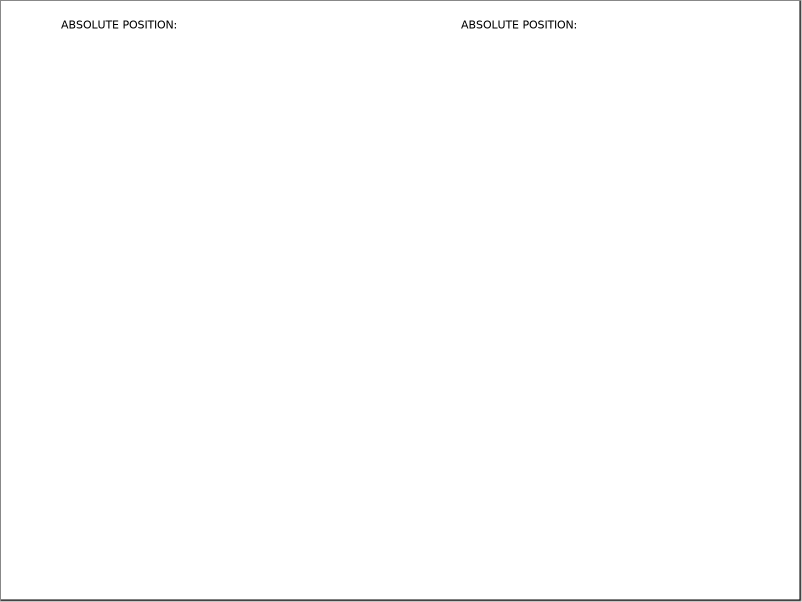
VISUALIZATION F51_Cam_Exchange  // 802x602
    Rectangle (0,0 800x600)
    Label (10,10 170x30), "ABSOLUTE POSITION:"
    Label (410,10 170x30), "ABSOLUTE POSITION:"
END_VISUALIZATION

(* stored: Version 1.1.0.1, ProductVersion 3.1.4022.7
   Visu F51_Cam_Exchange: Id {58aed0ed-8035-42bf-aefb-43119de631c0} *)
